{attribute 'qualified_only'}
VAR_GLOBAL
	bRemotePosted: BOOL := FALSE;
	bLocalGot: BOOL:= FALSE;
	blocalUpdated: BOOL:= TRUE;
	bMeasure: BOOL;
	aReadStruct : stData;
END_VAR

(* stored: Version 1.1.0.1, ProductVersion 3.1.4024.4
   GVL GlobalData: Id {3dca4ac0-a2c9-4424-81d1-723d81d6bac9} *)
